// TwinCAT 3 PLC project Untitled1
// ProgramVersion: 3.1.4026.16
// libraries:
//   Tc2_Standard, * (Beckhoff Automation GmbH)
//   Tc2_System, * (Beckhoff Automation GmbH)
// project tree:
//   / PlcTask.TcTTO
//   POUs/ fb_dancer.TcPOU, fb_motor.TcPOU, MAIN.TcPOU, fb_PID.TcPOU

CONFIGURATION Untitled1
    RESOURCE PLC ON TwinCAT3
        TASK PlcTask(INTERVAL := T#10ms, PRIORITY := 20);
        PROGRAM MAIN WITH PlcTask : MAIN;
    END_RESOURCE
END_CONFIGURATION

// ---- POUs/MAIN.TcPOU
PROGRAM MAIN
VAR
	r_targetPercent : REAL := 50;
	r_dancerPercent: REAL;
	r_accumulated_material_cm : REAL := 0;
	
	r_pid_Kp : REAL := -10;
	r_pid_Ki : REAL := -0.02;
	r_pid_Kd : REAL := -0.005;
	
	fb_motor : fb_motor;
	r_motorRPM : REAL;
	
	r_out_material_cm : REAL;
	r_in_material_cm : REAL;
	
	fb_dancer : fb_dancer;
	
	fb_PID: fb_PID;
	
	r_PID : REAL;
	r_P : REAL;
	r_I: REAL;
	r_D : REAL;
	
	r_Time : REAL;
	r_t : REAL;
	r_Kt : REAL := 5;
END_VAR

fb_motor(
	r_RPM := r_motorRPM,
	r_Radius := 20,
	r_dt := 0.01,
	r_out_cm => r_out_material_cm);

r_Time := r_Time + 0.01;

r_t := r_Time * r_Kt;
r_in_material_cm := 4*(20 + SIN(r_t) + SIN((r_t - 2.5) * 0.5)*2 + SIN((r_t + 1)*1.5)*1.33);

fb_dancer(
	r_in_cm := r_in_material_cm,
	r_out_cm := r_out_material_cm,
	r_dt := 0.01,
	r_accumulation => r_accumulated_material_cm,
	r_dancerPercent => r_dancerPercent);

fb_PID(
	r_ActVal:= r_dancerPercent, 
	r_SetVal:= r_targetPercent, 
	r_Kp:= r_pid_Kp, 
	r_Ki:= r_pid_Ki, 
	r_Kd:= r_pid_Kd, 
	r_dt:= 0.001, 
	r_maxValue := 100,
	r_minValue := -100,
	r_SampleRate := 1,
	r_PID=> r_PID, 
	r_P=> r_P, 
	r_I=> r_I, 
	r_D=> r_D);

r_motorRPM := LIMIT(0, r_motorRPM + r_PID, 160);

END_PROGRAM

// ---- POUs/fb_motor.TcPOU
FUNCTION_BLOCK fb_motor
VAR_INPUT
	r_RPM : REAL;
	r_Radius : REAL;
	r_dt : REAL;
END_VAR
VAR_OUTPUT
	r_out_cm : REAL;
END_VAR
VAR
	pi : REAL := 3.14159;
END_VAR

r_out_cm := (2 * pi * r_Radius) * (r_RPM / 60);

END_FUNCTION_BLOCK

// ---- POUs/fb_dancer.TcPOU
FUNCTION_BLOCK fb_dancer
VAR_INPUT
	r_in_cm: REAL;
	r_out_cm: REAL;
	r_dt : REAL;
END_VAR
VAR_OUTPUT
	r_accumulation : REAL;
	r_dancerPercent  : REAL;
END_VAR
VAR
END_VAR

r_accumulation := r_accumulation + ((r_in_cm - r_out_cm) * r_dt);
r_dancerPercent := LIMIT(0, r_accumulation / 5, 100);

END_FUNCTION_BLOCK

// ---- POUs/fb_PID.TcPOU
FUNCTION_BLOCK fb_PID
VAR_INPUT
	r_ActVal : REAL;
	r_SetVal : REAL;
	r_Kp : REAL;
	r_Ki : REAL;
	r_Kd : REAL;
	r_dt : REAL;
	
	r_maxValue : REAL;
	r_minValue : REAL;
	
	r_SampleRate : REAL;
END_VAR
VAR_OUTPUT
	r_PID : REAL;
	r_P : REAL;
	r_I : REAL;
	r_D : REAL;
END_VAR
VAR
	r_Error : REAL;
	r_PrevError : REAL;
	i_ArraySize : INT := 20;
	r_ErrorHistory : ARRAY[1..20] OF REAL;
	i : INT;
	Kp: REAL;
	r_Sum : REAL;
	r_SampleCounter : INT := 0;
END_VAR

r_PrevError := r_Error;
r_Error := r_SetVal - r_ActVal;

r_SampleCounter := r_SampleCounter + 1;

IF r_SampleCounter = r_SampleRate THEN
	r_SampleCounter := 0;
	FOR i := 1 TO i_ArraySize - 1 DO
		r_ErrorHistory[i+1] := r_ErrorHistory[i];
	END_FOR
	r_ErrorHistory[1] := r_Error;
END_IF 

FOR i := 1 TO i_ArraySize DO
	r_Sum := r_Sum + r_ErrorHistory[i];
END_FOR

r_P := r_Kp * r_Error;
r_I := r_Ki * r_Sum * r_dt;
r_D := r_Kd * ((r_Error - r_PrevError) / r_dt);

r_PID := LIMIT(r_minValue, r_P + r_I + r_D, r_maxValue);

END_FUNCTION_BLOCK
